// TIA Portal V19 export
ORGANIZATION_BLOCK "Main"   // OB1, LAD, ProgramCycle
TITLE = "Main Program Sweep (Cycle)"
{ S7_Optimized_Access := 'TRUE' }
// stored: SetENOAutomatically false
   VAR_INPUT
      Initial_Call : Bool;   // Initial call of this OB
      Remanence : Bool;   // =True, if remanent data are available
   END_VAR
BEGIN

REGION Network 1
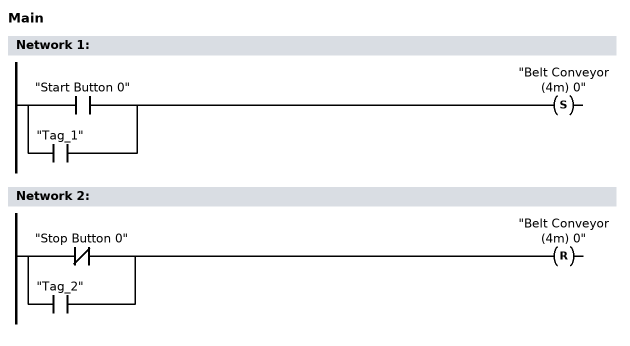
   RUNG wire#powerrail
      Contact( "Start Button 0" )
      wire#w1
      S_Coil( "Belt Conveyor (4m) 0" )
   END_RUNG
   RUNG wire#powerrail
      Contact( "Tag_1" )
   END_RUNG wire#w1
   // the same network as SCL:
   IF "Start Button 0" OR "Tag_1" THEN "Belt Conveyor (4m) 0" := TRUE; END_IF;
END_REGION

REGION Network 2
   RUNG wire#powerrail
      I_Contact( "Stop Button 0" )
      wire#w1
      R_Coil( "Belt Conveyor (4m) 0" )
   END_RUNG
   RUNG wire#powerrail
      Contact( "Tag_2" )
   END_RUNG wire#w1
   // the same network as SCL:
   IF NOT "Stop Button 0" OR "Tag_2" THEN "Belt Conveyor (4m) 0" := FALSE; END_IF;
END_REGION
END_ORGANIZATION_BLOCK
